// TwinCAT 3 PLC project ph_lv1_Communication
// Title: tclib_ph_lv1_generic_communication_interface
// Company: Poh
// Author: Poh
// ProjectVersion: 0.1.1.0
// ProgramVersion: 3.1.4020.1
// libraries:
//   tclib_ph_lv0, * (Poh)
// project tree:
//   Lv1_Communication/Class Interface/ IFC_GENERIC_COMMUNICATION_INTERFACE.TcIO
//   Lv1_Communication/Data Definition/ S_GCI_CONFIG.TcDUT, T_COMMHANDLE.TcDUT
//   Project Information/ F_GetCompany.TcPOU, F_GetTitle.TcPOU
//   Version/ Global_Version.TcGVL
// (motion and I/O tree: see PLC project ph_lv0)
// real-time tasks:
//   TASK PlcTask: cycle T#10ms, priority 20, ADS port 350

// ---- Lv1_Communication/Data Definition/S_GCI_CONFIG.TcDUT
(*
	Y:2016		M:05	D:20
	GENERIC COMMUNICATION CONFIGURATION 
*)
TYPE S_GCI_CONFIG :
STRUCT
	//25 byte data for storing communication address, and/or additional configurations
		Comm_Handle	: T_COMMHANDLE;
	//Generic data pointer to communication data buffer
		P_Data		: PVOID;
	//Communication data size
		Data_Size	: UDINT;
END_STRUCT
END_TYPE

// ---- Lv1_Communication/Data Definition/T_COMMHANDLE.TcDUT
TYPE T_COMMHANDLE : ARRAY[0..255] OF USINT; END_TYPE

// ---- Version/Global_Version.TcGVL
{attribute 'TcGenerated'}
// This function has been automatically generated from the project information.
VAR_GLOBAL CONSTANT
	{attribute 'const_non_replaced'}
	{attribute 'linkalways'}
	stLibVersion_tclib_ph_lv1_generic_communication_interface : ST_LibVersion := (iMajor := 0, iMinor := 1, iBuild := 1, iRevision := 0, sVersion := '0.1.1.0');
END_VAR

// ---- Lv1_Communication/Class Interface/IFC_GENERIC_COMMUNICATION_INTERFACE.TcIO
(*
	Y:2016	M:05	D:20
	T:INTERFACE		N:GENERIC COMMUNICATION INTERFACE
*)
INTERFACE IFC_GENERIC_COMMUNICATION_INTERFACE

METHOD Close_Connection : RETURN_CODE
VAR_INPUT
END_VAR
END_METHOD

METHOD Create_Handle : RETURN_CODE
VAR_INPUT
	Configuration 	: POINTER TO S_GCI_CONFIG;
	OUT_HANDLE		: POINTER TO UDINT;
END_VAR
END_METHOD

METHOD Open_Connection : RETURN_CODE
VAR_INPUT
	CONNECTION_INFO : POINTER TO S_GCI_CONFIG;
END_VAR
END_METHOD

METHOD Read : RETURN_CODE
VAR_INPUT
	Configuration : POINTER TO S_GCI_CONFIG;
END_VAR
END_METHOD

METHOD Release_Handle : RETURN_CODE
VAR_INPUT
	IN_HANDLE : POINTER TO UDINT;
END_VAR
END_METHOD

METHOD Write : RETURN_CODE
VAR_INPUT
	Configuration : POINTER TO S_GCI_CONFIG;
END_VAR
END_METHOD

END_INTERFACE

// ---- Project Information/F_GetCompany.TcPOU
// This function has been automatically generated from the project information.
{attribute 'signature_flag' := '1073741824'}
{attribute 'TcGenerated'}
FUNCTION F_GetCompany : WSTRING
VAR_INPUT
	
END_VAR

F_GetCompany := "Poh";

END_FUNCTION

// ---- Project Information/F_GetTitle.TcPOU
// This function has been automatically generated from the project information.
{attribute 'signature_flag' := '1073741824'}
{attribute 'TcGenerated'}
FUNCTION F_GetTitle : WSTRING
VAR_INPUT
	
END_VAR

F_GetTitle := "tclib_ph_lv0";

END_FUNCTION
